FUNCTION_BLOCK FB_SendCurrentAngle
VAR_INPUT
	CurrentAngle : LREAL;
END_VAR
VAR_OUTPUT
END_VAR
VAR
	TxMessage : EXTCANQUEUE;
	i : INT;
	CurrentAngle_Values : ARRAY[0..1] OF BYTE;
END_VAR
VAR_IN_OUT
	CAN_OUTPUTS : CANTXQUEUESTRUCT_E_32;
	CAN_INPUTS : CANRXQUEUESTRUCT_E_32;
END_VAR

CurrentAngle_Values[1] := INT_TO_BYTE(LREAL_TO_INT(CurrentAngle) AND 16#FF);
CurrentAngle_Values[0] := INT_TO_BYTE(SHR(LREAL_TO_INT(CurrentAngle), 8) AND 16#FF);


TxMessage.cobId := 1100;
TxMessage.length := 2;
FOR i := 0 TO 1 DO 
		TxMessage.data[i] := CurrentAngle_Values[i];
END_FOR
CAN_OUTPUTS.TxMessages[1] := TxMessage;
//CAN_OUTPUTS.NoOfTxMessages := 1;


(*
TxMessage.cobId := 1100;
TxMessage.length := 2;
FOR i := 0 TO 1 DO 
			TxMessage.data[i] := CurrentAngle_Values[i];
END_FOR
CAN_OUTPUTS.TxMessages[0] := TxMessage;
CAN_OUTPUTS.TxCounter := CAN_INPUTS.TxCounter + 1;
*)

END_FUNCTION_BLOCK

(* stored: Version 1.1.0.1
   POU FB_SendCurrentAngle: Id {7141db5d-6b5f-4edd-ac1f-fa7f9535ab81}, SpecialFunc None *)
